TYPE "MES_Msg_Receive_Topic3xx_Err"
VERSION : 0.1
// Block: MES_Msg_Receive_Topic3xx_Err
   STRUCT
      Recive_MSG300 : "MES_Err_&_Msg";
      Recive_MSG301 : "MES_Err_&_Msg";
   END_STRUCT;

END_TYPE
